// TwinCAT 3 PLC project Stamp
// ProgramVersion: 3.1.4026.11
// libraries:
//   Tc2_Standard, * (Beckhoff Automation GmbH)
//   Tc2_System, * (Beckhoff Automation GmbH)
//   [Resi4MPM], * (Jan Wilch)
//   [xPPU], * (Jan Wilch)
// project tree:
//   / HardwareContainer.TcPOU, MAIN.TcPOU, PlcTask.TcTTO
// (motion and I/O tree: see PLC project crane)
// real-time tasks:
//   TASK PlcTask: cycle T#10ms, priority 20, ADS port 350
//   TASK PlcTask1: cycle T#10ms, priority 23, ADS port 351
//   TASK PlcTask2: cycle T#10ms, priority 22, ADS port 352
//   TASK PlcTask3: cycle T#10ms, priority 21, ADS port 353
// variable links:
//   Stamp/Stamp Instance <-> Device (EtherCAT)/BK2&3 (EK1100)/2&3.10 (EL2004)
//     PlcTask Outputs/MAIN.m_container.m_stamp.m_slidingCylinder.DO_Extend <-> Channel 1/Output
//     PlcTask Outputs/MAIN.m_container.m_stamp.m_slidingCylinder.DO_Retract <-> Channel 2/Output
//     PlcTask Outputs/MAIN.m_container.m_stamp.m_stampingCylinder.DO_Extend <-> Channel 3/Output
//     PlcTask Outputs/MAIN.m_panelMgr.DO_GreenLight <-> Channel 4/Output
//   Stamp/Stamp Instance <-> Device (EtherCAT)/BK2&3 (EK1100)/2&3.11 (EL2004)
//     PlcTask Outputs/MAIN.m_panelMgr.DO_WhiteLight <-> Channel 1/Output
//   Stamp/Stamp Instance <-> Device (EtherCAT)/BK2&3 (EK1100)/2&3.16 (EL4102)
//     PlcTask Outputs/MAIN.m_container.m_stamp.m_pressureValve.AO_SetPressure <-> Channel 2/Output
//   Stamp/Stamp Instance <-> Device (EtherCAT)/BK2&3 (EK1100)/2&3.2 (EL1004)
//     PlcTask Inputs/MAIN.m_container.m_stamp.m_slidingCylinder.DI_Extended <-> Channel 2/Input
//     PlcTask Inputs/MAIN.m_container.m_stamp.m_slidingCylinder.DI_Retracted <-> Channel 3/Input
//     PlcTask Inputs/MAIN.m_container.m_stamp.m_stampingCylinder.DI_Retracted <-> Channel 4/Input
//     PlcTask Inputs/MAIN.m_panelMgr.DI_ModeSwitch <-> Channel 1/Input
//   Stamp/Stamp Instance <-> Device (EtherCAT)/BK2&3 (EK1100)/2&3.3 (EL1004)
//     PlcTask Inputs/MAIN.m_container.m_stamp.m_presenceSensor.DI_WPDetected <-> Channel 2/Input
//     PlcTask Inputs/MAIN.m_container.m_stamp.m_stampingCylinder.DI_Extended <-> Channel 1/Input
//   Stamp/Stamp Instance <-> Device (EtherCAT)/BK2&3 (EK1100)/2&3.7 (EL1004)
//     PlcTask Inputs/MAIN.m_panelMgr.DI_EStopBtn <-> Channel 3/Input
//     PlcTask Inputs/MAIN.m_panelMgr.DI_StartBtn <-> Channel 4/Input
//   Stamp/Stamp Instance <-> Device (EtherCAT)/BK4 (EK1100)/4.3 (EL1004)
//     PlcTask Inputs/MAIN.m_container.m_stamp.m_slidingCylinder.DI_BoundaryPressure <-> Channel 2/Input
//   Stamp/Stamp Instance <-> Device (EtherCAT)/BK4 (EK1100)/4.4 (EL1004)
//     PlcTask Inputs/MAIN.m_container.m_stamp.m_stampingCylinder.DI_BoundaryPressure <-> Channel 4/Input
//   Stamp/Stamp Instance <-> Device (EtherCAT)/BK4 (EK1100)/4.6 (EL1004)
//     PlcTask Inputs/MAIN.m_container.m_stamp.m_stampingCylinder.DI_BoundaryFlowPressure <-> Channel 1/Input
//   Stamp/Stamp Instance <-> Device (EtherCAT)/BK4 (EK1100)/4.9 (EL3064)
//     PlcTask Inputs/MAIN.m_container.m_stamp.m_stampingCylinder.AI_PressureSensor <-> AI Standard Channel 2/Value
//   Stamp/Stamp Instance <-> Device (EtherCAT)/BK4 (EK1100)/Term 90 (EL3058)
//     PlcTask Inputs/MAIN.m_container.m_stamp.m_slidingCylinder.AI_PositionTransmitter <-> AI Standard Channel 3/Value
//     PlcTask Inputs/MAIN.m_container.m_stamp.m_stampingCylinder.AI_PositionTransmitter <-> AI Standard Channel 4/Value

CONFIGURATION Stamp
    RESOURCE PLC ON TwinCAT3
        TASK PlcTask(INTERVAL := T#10ms, PRIORITY := 23);
        PROGRAM MAIN WITH PlcTask : MAIN;
    END_RESOURCE
END_CONFIGURATION

// ---- MAIN.TcPOU
PROGRAM MAIN
VAR CONSTANT
	IGNORE_DEFINITION: BOOL := TRUE;
END_VAR
VAR
	m_errorManager: ErrorManager;
	m_services: ServiceContainer(ADR(m_errorManager));
	
	m_panelMgr: PanelManager(
		m_services.PtrStateTracker,
		EProcessVariables.Pnl_Stamp_Start,
		0,
		EProcessVariables.Pnl_Stamp_Mode,
		EProcessVariables.Pnl_Stamp_EStop,
		0);
	
	// instantiate machine behavior model
	m_container: HardwareContainer(
		m_services.PtrStateTracker, 
		m_services.PtrProcessManager, 
		ADR(m_errorManager));
	
	m_modes: MachineModes(ADR(m_services), ADR(m_panelMgr));
	
	m_appObservation: ARRAY[EProcessVariables.OpMode_Stamp..EProcessVariables.OpMode_Stamp] OF SValue;

	// TESTING
// 	m_lscConnected: BOOL;
// 	m_craneConnected: BOOL;
// 	m_stackConnected: BOOL;
// 	m_stampConnected: BOOL;
END_VAR

// process state observation
m_appObservation[EProcessVariables.OpMode_Stamp].DataType := EDataType.string_t;
m_appObservation[EProcessVariables.OpMode_Stamp].Value.String_t := m_modes.SFCCurrentStep;
m_appObservation[EProcessVariables.OpMode_Stamp].Defined := TRUE;

// cylic service updates
m_services.PtrStateTracker^.CyclicUpdateStatus(IGNORE_DEFINITION, m_appObservation);
m_services.PtrProcessManager^.CyclicManageBehavior();

// main state machine
m_modes();

// TESTING
// IF m_services.PtrStateTracker^.GetString(EProcessVariables.OpMode_LSC) <> '' THEN
// 	m_lscConnected := TRUE;
// END_IF
// IF m_services.PtrStateTracker^.GetString(EProcessVariables.OpMode_Stack) <> '' THEN
// 	m_stackConnected := TRUE;
// END_IF
// IF m_services.PtrStateTracker^.GetString(EProcessVariables.OpMode_Stamp) <> '' THEN
// 	m_stampConnected := TRUE;
// END_IF
// IF m_services.PtrStateTracker^.GetString(EProcessVariables.OpMode_Crane) <> '' THEN
// 	m_craneConnected := TRUE;
// END_IF

END_PROGRAM

// ---- HardwareContainer.TcPOU
FUNCTION_BLOCK HardwareContainer
VAR
	// hardware control POUs
	m_stamp: Stamp;
	m_indic: ActivityIndicator(i_signalProcVar := EProcessVariables.Test_StampFree);
	
	// products
	{attribute 'OPC.UA.DA' := '1'}
	{attribute 'OPC.UA.DA.Access' := '1'}
	m_stampWP: xPPUProduct(EProcessVariables.Stamp_ProductType, EProcessVariables.Stamp_ProductStamped);
	
	// hardware observation (if not included in hardware control)
	m_observeStamp: ObserveStamp(ADR(m_stamp), ADR(m_stampWP));
	
	// control primitives
	m_stampStamp: Stamp_StampWorkpiece(ADR(m_stamp));
	m_delay: Delay;
	m_indicCP_Stamp: IndicateActivity(i_id := EPrimitives.Gen_IndicateActive_Stamp, i_ptrIndicator := ADR(m_indic));
	m_forceVal_Stamp: ForceProcessVariable(i_id := EPrimitives.Gen_ForceVariable_Stamp);
	
	// module sequences
END_VAR

METHOD FB_init : BOOL
VAR_INPUT
	bInitRetains : BOOL; // if TRUE, the retain variables are initialized (warm start / cold start)
	bInCopyCode : BOOL;  // if TRUE, the instance afterwards gets moved into the copy code (online change)

	i_ptrStateTracker: POINTER TO StateTracker;
	i_ptrProcessManager: POINTER TO ProcessManager;
	
	i_ptrErrorManager: POINTER TO ErrorManagerBase;
END_VAR
m_stampStamp.ProvideServices(i_ptrProcessManager, i_ptrStateTracker);
m_delay.ProvideServices(i_ptrProcessManager, i_ptrStateTracker);
m_indicCP_Stamp.ProvideServices(i_ptrProcessManager, i_ptrStateTracker);
m_forceVal_Stamp.ProvideServices(i_ptrProcessManager, i_ptrStateTracker);

// provide Behaviors to the Process Manager
i_ptrProcessManager^.AddPrimitive(ADR(m_stampStamp));
i_ptrProcessManager^.AddPrimitive(ADR(m_delay));
i_ptrProcessManager^.AddPrimitive(ADR(m_indicCP_Stamp));
i_ptrProcessManager^.AddPrimitive(ADR(m_forceVal_Stamp));

// provide observations to the Process Manager
i_ptrStateTracker^.AddObservation(ADR(m_observeStamp));
i_ptrStateTracker^.AddObservation(ADR(m_indic));

// provide workpieces to the Process Manager
i_ptrStateTracker^.RegisterLocalProduct(EProducts.stamp_product, ADR(m_stampWP));
END_METHOD

END_FUNCTION_BLOCK
